TYPE INTERNAL ST_CylinderInfo :
STRUCT
	sensorHP			: BOOL;
	sensorWP			: BOOL;
END_STRUCT
END_TYPE

(* stored: Version 1.1.0.1, ProductVersion 3.1.4026.17
   DUT ST_CylinderInfo: Id {d47935cc-7287-0c1e-0aef-c0a2bee02841} *)
